FUNCTION Convert_DWORD_TO_LREAL : Hresult
VAR_INPUT
	in : DWORD;
	out : REFERENCE TO LREAL;
END_VAR
VAR
	converted : LREAL;
END_VAR

converted := DWORD_TO_LREAL(in);

IF (LREAL_TO_DWORD(converted) <> in) THEN
	Convert_DWORD_TO_LREAL := INCOMPATIBLE;
	RETURN;
END_IF

out := converted;

END_FUNCTION

(* stored: Version 1.1.0.1, ProductVersion 3.1.4024.12
   POU Convert_DWORD_TO_LREAL: Id {7c8c2dd4-5540-4063-b0e2-1caaec4774ba}, SpecialFunc None *)
